(*
	Basic device with extended interface:
	nControl BYTE: From TwinCAT >>> To Unity
	nStatus BYTE: FROM Unity >>> TO TwinCAT	
	nControlData LWORD: From TwinCAT >>> To Unity
	nStatusData LWORD: FROM Unity >>> TO TwinCAT	
*)
FUNCTION_BLOCK FB_DeviceLWord EXTENDS FB_LinkDataLWord
VAR_INPUT		
	nControl  			: BYTE;
	nControlData  		: LWORD;
END_VAR

VAR_OUTPUT
	nStatus  			: BYTE;
	nStatusData  		: LWORD;
END_VAR

SUPER^();
Control := nControl;
ControlData := nControlData;
nStatus := Status;
nStatusData := StatusData;

END_FUNCTION_BLOCK

(* stored: Version 1.1.0.1, ProductVersion 3.1.4024.12
   POU FB_DeviceLWord: Id {ebc2de75-3ab5-0d8f-0ee5-fb01e22b2b7a}, SpecialFunc None *)
